GLOBALCONSTANTS DefaultPool_PWM_Bargraph (* Bargraph geometry and scale constants (Length, ScalePx, Min, Max, Type) *)
  PACKAGE Uebungen::const::UT::PWM;
  VAR_GLOBAL CONSTANT
    LinearBargraph_ScalePx : REAL := 0.0586009034;
    LinearBargraph_LengthPx : REAL := 480.0;
    LinearBargraph_Min : REAL := 0.0;
    LinearBargraph_Max : REAL := 8191.0;
    LinearBargraph_Type : USINT := 3;
  END_VAR
END_GLOBALCONSTANTS
